TYPE ST_MESSAGE_CTRL :
STRUCT
  Cmd         : E_MESSAGE_CTRL;
END_STRUCT
END_TYPE

(* stored: Version 1.1.0.1, ProductVersion 3.1.4026.13
   DUT ST_MESSAGE_CTRL: Id {5f449fa6-064f-4819-8cc9-fae3a381a7a7} *)
